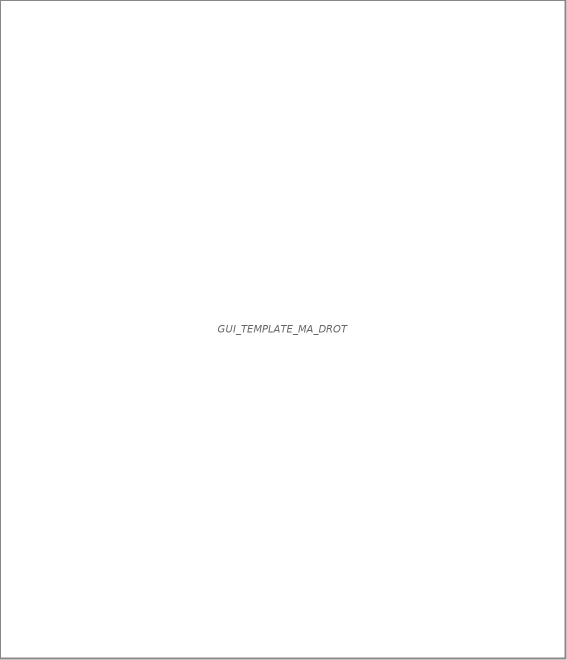
VISUALIZATION GUI_MA_DROT  // 567x660
    Frame (0,0 565x658)
        shows GUI_TEMPLATE_MA_DROT(m_DeviceName := 'DROT', m_Instance := MAIN.drot)
END_VISUALIZATION

(* stored: Version 1.1.0.1, ProductVersion 3.1.4022.16
   Visu GUI_MA_DROT: Id {27c61d1d-d13b-4618-a191-c7fda807e85e} *)
